FUNCTION_BLOCK T_AdsReadWrite IMPLEMENTS I_Executable
VAR
   logger : I_Logger;
	_readWriteOpts : ST_AdsReadWriteOptions;
	
   readWrite : ADSRDWRT;

   state, prevState : (
      IDLE,
      REQUEST,
      WAIT_FOR_RESPONSE,
      DONE_STATE,
      ERROR_STATE
   );

   lastErrorId : UDINT;

END_VAR
VAR CONSTANT
   NO_ERR : UDINT := 0;
   LOG_DEBUG : DWORD := 0;
   LOG_INFO : DWORD := ADSLOG_MSGTYPE_HINT;
   LOG_WARNING : DWORD := ADSLOG_MSGTYPE_WARN;
   LOG_ERROR : DWORD := ADSLOG_MSGTYPE_ERROR;
END_VAR

CASE state OF

   IDlE:
      IsEntryActionAndLog();

   REQUEST:
      IsEntryActionAndLog();
		
      lastErrorId := NO_ERR;
      readWrite.WRTRD := TRUE;
      state := WAIT_FOR_RESPONSE;

   WAIT_FOR_RESPONSE:
      IsEntryActionAndLog();

      IF readWrite.ERR THEN
         state := ERROR_STATE;

      ELSIF NOT readWrite.BUSY THEN
         state := DONE_STATE;

      END_IF

   DONE_STATE:
      IsEntryActionAndLog();

   ERROR_STATE:
      IF IsEntryActionAndLog() THEN
         lastErrorId := readWrite.ERRID;
			
      END_IF

END_CASE

readWrite.WRTRD R= NOT Busy;
readWrite();

PROPERTY Busy : BOOL
GET
Busy := 
	NOT Done 
	AND NOT Error 
	AND state <> IDLE;
END_GET
END_PROPERTY

PROPERTY Done : BOOL
GET
Done := state = DONE_STATE;
END_GET
END_PROPERTY

PROPERTY Error : BOOL
GET
Error := state = ERROR_STATE;
END_GET
END_PROPERTY

METHOD PRIVATE IsEntryActionAndLog : BOOL
IsEntryActionAndLog := prevState <> state;

// useful to debug state transitions. to avoid "chatter" LogFramework should have runtime log level switches 
// i.e. https://github.com/Intecre/twincat-utils/tree/master/IntecreUtilities/IntecreUtilities/IntecreUtilities/Utilities/Logger
// see also https://github.com/Intecre/twincat-utils/blob/master/IntecreUtilities/IntecreUtilities/IntecreUtilities/Utilities/T_NamedBase.TcPOU
ToLog(
	Msg := CONCAT(CONCAT(TO_STRING(prevState), ' transition to state '), TO_STRING(state)), 
	LogLevel:= LOG_DEBUG
);

prevState := state;
END_METHOD

METHOD PUBLIC SetLogger
VAR_INPUT
	logger : I_Logger;
END_VAR
THIS^.logger := logger;
END_METHOD

METHOD PRIVATE ToLog
VAR_INPUT
	Msg : STRING(255);
	LogLevel : DWORD; // generic level, can be mapped to logging framework
END_VAR
IF logger = 0 THEN
	RETURN;
	
END_IF

logger.ToLog(Msg, LogLevel);
END_METHOD

METHOD TryRequest : BOOL
VAR_INPUT
	readWriteOptions : ST_AdsReadWriteOptions;
END_VAR
VAR_OUTPUT
	status : I_Executable;
END_VAR
VAR CONSTANT
	NO_HANDLE : DWORD := 0;
END_VAR
IF Busy THEN
	ToLog('Cannot TryRequest as Busy', LOG_WARNING);
	RETURN;
	
END_IF

_readWriteOpts := readWriteOptions;
readWrite(
	NETID := F_GetAmsNetId(_readWriteOpts.AdsAddress.netId),
	PORT := _readWriteOpts.AdsAddress.port,
	IDXGRP := _readWriteOpts.IndexGroup,
	IDXOFFS := _readWriteOpts.IndexOffset,
	WRITELEN := _readWriteOpts.WriteParams.cbLen,
	SRCADDR := _readWriteOpts.WriteParams.pData,
	READLEN := _readWriteOpts.ReadParams.cbLen,
	DESTADDR := _readWriteOpts.ReadParams.pData,
	TMOUT := _readWriteOpts.Timeout
);

state := REQUEST;

TryRequest := TRUE;
status := THIS^;
END_METHOD

END_FUNCTION_BLOCK

(* stored: Version 1.1.0.1, ProductVersion 3.1.4024.9
   POU T_AdsReadWrite: Id {9e332780-0c6d-4776-8b7a-c762dffc295f}, SpecialFunc None
   Property Busy: Id {b532a871-df3e-4141-8e14-4ecf6fc04f0d}
   Get Get: Id {9c3b3619-f8b0-4210-ab35-a9e3fdd54faa}
   Property Done: Id {c64c9238-f6d1-4626-8cce-31f6f5c94936}
   Get Get: Id {265a5a66-9a59-4b7e-b132-dd6369ae7cfe}
   Property Error: Id {92c5d5bf-0374-4ca5-ad14-dfacf66780c5}
   Get Get: Id {8275ad9a-0b78-4d5b-bd8d-7fe1b2124449}
   Method IsEntryActionAndLog: Id {6dfd938b-ee7d-4b0f-a850-c29f6b8ffda3}
   Method SetLogger: Id {8f9a6c80-acd6-46c2-ad3f-f984d96aeb61}
   Method ToLog: Id {3345ce33-591b-47dc-9154-285ecdd50956}
   Method TryRequest: Id {2347141d-ee4b-4e78-a06d-f5c6ab63ca1b} *)
